//==================================================================================================
//							Beckhoff Automation Poland
//									18.04.2018
//	Struktura zawierajaca I/O odpowiedniego bloku
//  v1.0	|| TC v 3.1.4022.16		|| - pierwsza wersja
//==================================================================================================
TYPE ST_MCMoveModuloIO:
STRUCT
	bExecute						: BOOL;								// Rising edge executes cmd
	lrPosition						: LREAL;
	lrVelocity						: LREAL;
	lrAcceleration					: LREAL;
	lrDeceleration					: LREAL;
	lrJerk							: LREAL;
	eDirection						: Tc2_MC2.MC_Direction 		:= MC_Positive_Direction; // MC_Positive_Direction := 1, MC_Shortest_Way, MC_Negative_Direction, MC_Current_Direction
	eBufferMode						: Tc2_MC2.MC_BufferMode;
	stOptions						: Tc2_MC2.ST_MoveOptions;
	bDone							: BOOL;
	bBusy							: BOOL;
	bActive							: BOOL;
	bCommandAborted					: BOOL;
	bError							: BOOL;
	udiErrorID						: UDINT;
END_STRUCT
END_TYPE

(* stored: Version 1.1.0.1, ProductVersion 3.1.4026.13, FileIdentifier e96b6e6844c2678b1521d3069747de98636aea25, FileSignature 3e961e7924c32bdee1b841c3f552704d5c61af33a1c9a35498e81ecc6f4c3e7d8d10c56aa32bbb4f3d7d78dd5572eb4f946fe948ba356b0b0e5a40a38d6f01d3f54d6a8d75b7e81401217ea77a467645280969616ec3c5d6a3e94296d3d4c25b6fa44e34c22b83920a5515fb8064055bc33c995d38e1649b1a2a40dd1969b9666c87ee426e61e26e1a3e4b05ab42b96a3a0bc9b9df3f705c27ed8f38b08da52b17947b703963c09e143a2c31e6c3b9b470366a455ddea6e343bd8ff53f36b357aaf7663a228d92c19f8cda7bc7e1084d14d92bb070fcf143781d51bcc97f524adca5e25fbda1004c278eca4e3159236b9cf4d5b85164f72e51b77eea3534413a
   DUT ST_MCMoveModuloIO: Id {db103db5-6b32-497f-992d-b8cf8d9dbf33} *)
